(* CoDeSys 2.3 export: PLC_PRG.EXP *)

(* POU PLC_PRG, ST *)
PROGRAM PLC_PRG
VAR
	firstLoop:BOOL;
	test:INT;

	Attic:Attic;
	Bathroom_pietro:Bathroom_pietro;
	E_gabinet:E_gabinet;
	Garderoba:Garderoba;
	Hol_parter:Hol_parter;
	Julka:Julka;
	Kotlownia:Kotlownia;
	Lazienka_parter:Lazienka_parter;
	N_sypialnia:N_sypialnia;
	Przedpokoj_pietro:Przedpokoj_pietro;
	Salon:Salon;
	Zosia:Zosia;
	Taras:Taras;
	Studnia:Studnia;

	LockMode:LockMode;

END_VAR
IF NOT firstLoop THEN
	firstLoop:=1;
	start();
END_IF

lockMode();

attic();
bathroom_pietro();
e_gabinet();
garderoba();
hol_parter();
julka();
kotlownia(presenceDetection:=bathroom_pietro.presenceDetection XOR lazienka_parter.presenceDetection XOR salon.kuchniaPresenceDetection );
lazienka_parter();
n_sypialnia();
przedpokoj_pietro();
salon();
zosia();
taras();
studnia();

clock1secImpulse := 0;
clock01secImpulse:=0;
test := test + 1;
END_PROGRAM
